# EPICS substitutions: epics/m-epics-eemcu/eemcuApp/Db/Sim8-extra-m4.substitutions
file "eemcu-extra.template"
{
pattern
{P,      M,    R,   PORT, ADDR, PREC, HOMEPROC}
{IOC:,   m4, m4-,   MCU1,    4, 3,    3}
}
